PROGRAM MAIN_Fast
VAR
	fbGetCurTaskIdx 			: GETCURTASKINDEX;
	bFirstCycle					: BOOL;
//	For temperature feedback linearisation
	fbLinInterpolation			: FB_LIN_INTERPOLATION;
END_VAR


// =========================================================
	// Get plc task first cycle flag	
fbGetCurTaskIdx(); 
bFirstCycle:= _TaskInfo[fbGetCurTaskIdx.index].FirstCycle;

IF bFirstCycle THEN
	;
END_IF

	// Temperature feedback linearisation	
fbLinInterpolation();	
fbLinInterpolation.M_Cyclic();

// =========================================================

END_PROGRAM

(* stored: Version 1.1.0.1
   POU MAIN_Fast: Id {f3aabdab-143e-4e78-8800-ab31e3e5df70}, SpecialFunc None *)
